FUNCTION_BLOCK ValveControl (* Basic Function Block Type *)
  (* Standard: 61499-2 *)
  (* Version 0.0, 9/14/2008, Horst Mayer, nxtControl GmbH, Template *)
  PACKAGE Main;
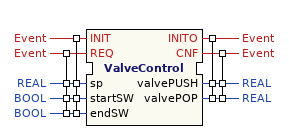
  EVENT_INPUT
    INIT WITH sp, startSW, endSW; (* Initialization Request *)
    REQ WITH sp, startSW, endSW; (* Normal Execution Request *)
  END_EVENT
  EVENT_OUTPUT
    INITO WITH valvePUSH, valvePOP; (* Initialization Confirm *)
    CNF WITH valvePUSH, valvePOP; (* Execution Confirmation *)
  END_EVENT
  VAR_INPUT
    sp : REAL;
    startSW : BOOL;
    endSW : BOOL;
  END_VAR
  VAR_OUTPUT
    valvePUSH : REAL;
    valvePOP : REAL;
  END_VAR
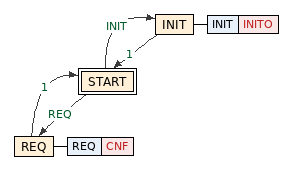
  EC_STATES
    START; (* Initial State *)
    INIT : INIT -> INITO; (* Initialization *)
    REQ : REQ -> CNF; (* Normal execution *)
  END_STATES
  EC_TRANSITIONS
    START TO INIT := INIT;
    INIT TO START := 1;
    START TO REQ := REQ;
    REQ TO START := 1;
  END_TRANSITIONS
  ALGORITHM INIT IN ST: (* Initialization algorithm *)
valvePOP := 0.0;
valvePUSH := 0.0;
  END_ALGORITHM
  ALGORITHM REQ IN ST: (* Normally executed algorithm *)
IF sp < 0.0 THEN
 IF startSW THEN
 	valvePOP := 0.0;
 ELSE
	 valvePOP := sp * -1.0;
 END_IF;
 valvePUSH := 0.0;
ELSIF sp > 0.0 THEN
 valvePOP := 0.0;
 IF endSW THEN
 	valvePUSH := 0.0;
 ELSE
 	valvePUSH := sp;
 END_IF;
ELSE
 valvePOP := 0.0;
 valvePUSH := 0.0;
END_IF;
  END_ALGORITHM
END_FUNCTION_BLOCK
